TYPE Visu_typ :
STRUCT
	
	MoveDirect_X		: LREAL;
	MoveDirect_Y		: LREAL;
	MoveDirect_Z 		: LREAL;

END_STRUCT
END_TYPE

(* stored: Version 1.1.0.1, ProductVersion 3.1.4024.11
   DUT Visu_typ: Id {2b0a5f95-68b2-4eb8-bf98-c32a10b5eac6} *)
